(* IEC 61131-3 sources: eCockpitGit/test_project/src/%F%00 Library/%F%Common Functions/%F%Module Value Conversion, 5 files *)

(* ---- %DUT%SModuleValueConversion3Point.st ---- *)
//Struct containing needed information to perform af 3 point calibration from a module value
// |**Version**|**Author**| **Date** |**Changes**
// | 1         | NSN      | 29-03-22 | Creation
TYPE SModuleValueConversion3Point :
STRUCT
	moduleUID		:AModuleUID;	//UID of module with value
	minValue		:UValue;		//Minimum value of conversion
	midValue		:UValue;		//Middle value of conversion
	maxValue		:UValue;		//Maximum value of conversion
END_STRUCT
END_TYPE

(* ---- %POU%FU_moduleValue3PointFromStruct.st ---- *)
//Reads a 3 point conversion struct from a reader
// |**Version**|**Author**| **Date** |**Changes**
// | 1         | NSN      | 29-03-22 | Creation
FUNCTION FU_moduleValue3PointFromStruct : BOOL
VAR_INPUT
	reader			:ITF_StructReaderBase;			//Reader
END_VAR
VAR_IN_OUT
	data			:SModuleValueConversion3Point;	//3 Point conversion struct
END_VAR
VAR
	module			:AModule;
END_VAR

(*%!%__DELIMITER__%!%*)
IF reader.valueType = EStructType.object THEN
	reader.enterObjectArray();
	IF reader.findKey(name:=GTSmall.Suid) <> EStructType.none THEN
		module						:=		GMod.modMan.getModuleByUID(modUID:=reader.readWord());
		IF module <> 0 THEN
			data.moduleUID			:=		module^._UID;
			IF reader.findKey(name:=GTSmall.Smin) <> EStructType.none THEN
				data.minValue		:=		FU_readUValue(reader:=reader,valueType:=module^.SYS_valueType);
			END_IF
			IF reader.findKey(name:=GTSmall.Smid) <> EStructType.none THEN
				data.midValue		:=		FU_readUValue(reader:=reader,valueType:=module^.SYS_valueType);
			END_IF
			IF reader.findKey(name:=GTSmall.Smax) <> EStructType.none THEN
				data.maxValue		:=		FU_readUValue(reader:=reader,valueType:=module^.SYS_valueType);
			END_IF
		END_IF
	END_IF
	reader.exitObjectArray();
END_IF

(* ---- %POU%FU_moduleValue3PointFromStructWithType.st ---- *)
//Reads a 3 point conversion struct from a reader
// |**Version**|**Author**| **Date** |**Changes**
// | 1         | NSN      | 29-03-22 | Creation
FUNCTION FU_moduleValue3PointFromStructWithType : BOOL
VAR_INPUT
	reader			:ITF_StructReaderBase;			//Reader
END_VAR
VAR_IN_OUT
	data			:SModuleValueConversion3Point;	//3 Point conversion struct
END_VAR

(*%!%__DELIMITER__%!%*)
IF reader.valueType = EStructType.object THEN
	reader.enterObjectArray();
	IF reader.findKey(name:=GTSmall.Suid) <> EStructType.none THEN
		data.moduleUID			:=		reader.readWord();
		IF reader.findKey(name:=GTSmall.Smin) = EStructType.tArray THEN
			FU_readUValueWithType(value=>data.minValue,reader:=reader);
		END_IF
		IF reader.findKey(name:=GTSmall.Smid) = EStructType.tArray THEN
			FU_readUValueWithType(value=>data.midValue,reader:=reader);
		END_IF
		IF reader.findKey(name:=GTSmall.Smax) = EStructType.tArray THEN
			FU_readUValueWithType(value=>data.maxValue,reader:=reader);
		END_IF
	END_IF
	reader.exitObjectArray();
END_IF

(* ---- %POU%FU_moduleValue3PointToStruct.st ---- *)
//Writes a 3 point conversion struct to a writer
// |**Version**|**Author**| **Date** |**Changes**
// | 1         | NSN      | 29-03-22 | Creation
FUNCTION FU_moduleValue3PointToStruct : BOOL
VAR_INPUT
	writer			:ITF_StructWriterBase;			//Writer
END_VAR
VAR_IN_OUT
	data			:SModuleValueConversion3Point;	//3 Point conversion struct
END_VAR
VAR
	module			:AModule;
	valueType		:EValueType;
END_VAR

(*%!%__DELIMITER__%!%*)
writer.objectStart(singleLine:=TRUE);
writer.addKey(name:=GTSmall.Suid);
writer.writeDint(value:=data.moduleUID);
module				:=		GMod.modMan.getModuleByUID(modUID:=data.moduleUID);
IF module <> 0 THEN
	valueType		:=		module^.SYS_valueType;
	writer.addKey(name:=GTSmall.Smin);
	FU_writeUValue(value:=data.minValue,valueType:=valueType,writer:=writer);
	writer.addKey(name:=GTSmall.Smid);
	FU_writeUValue(value:=data.midValue,valueType:=valueType,writer:=writer);
	writer.addKey(name:=GTSmall.Smax);
	FU_writeUValue(value:=data.maxValue,valueType:=valueType,writer:=writer);
END_IF
writer.structEnd();

(* ---- %POU%FU_moduleValue3PointToStructWithType.st ---- *)
//Writes a 3 point conversion struct to a writer
// |**Version**|**Author**| **Date** |**Changes**
// | 1         | NSN      | 29-03-22 | Creation
FUNCTION FU_moduleValue3PointToStructWithType : BOOL
VAR_INPUT
	writer			:ITF_StructWriterBase;			//Writer
END_VAR
VAR_IN_OUT
	data			:SModuleValueConversion3Point;	//3 Point conversion struct
END_VAR
VAR
	module			:AModule;
	valueType		:EValueType;
END_VAR

(*%!%__DELIMITER__%!%*)
writer.objectStart(singleLine:=TRUE);
writer.addKey(name:=GTSmall.Suid);
writer.writeDint(value:=data.moduleUID);
module				:=		GMod.modMan.getModuleByUID(modUID:=data.moduleUID);
IF module <> 0 THEN
	valueType		:=		module^.SYS_valueType;
	writer.addKey(name:=GTSmall.Smin);
	FU_writeUValueWithType(value:=data.minValue,valueType:=valueType,writer:=writer);
	writer.addKey(name:=GTSmall.Smid);
	FU_writeUValueWithType(value:=data.midValue,valueType:=valueType,writer:=writer);
	writer.addKey(name:=GTSmall.Smax);
	FU_writeUValueWithType(value:=data.maxValue,valueType:=valueType,writer:=writer);
END_IF
writer.structEnd();
